FUNCTION_BLOCK RunAoiInspectionV1 EXTENDS RunUnitSlave
VAR_INPUT
	ngBinReady : BOOL;
	ngCounter : POINTER TO UDINT;
END_VAR
VAR_OUTPUT
END_VAR
VAR
	//devices
	ngCylinder : POINTER TO RunCylinder; // normal close cylinder
	
	aoiOut1Done AT%I* : BOOL ; //done
	aoiOut2Grade AT%I* : BOOL ; //ok/ng
	
	aoiTrigger AT%Q* : BOOL;
	//internal
	
	commIdTrigger AT%Q* : DWORD;
	
	//
	serialNGCounter : INT;
END_VAR
VAR PERSISTENT
	serialNGGoal AT%M* : INT ;
END_VAR
VAR CONSTANT
	ERR_CONSECUTIVE_NG : DWORD := 8001;
END_VAR

SUPER^();

CASE outputState OF
	//--------------------------------
	//	Initialization TODO, (Light on?)
	//--------------------------------	
	eSpecialStates.INITIAL_BEGIN:	
		bSerialTransition := ngCylinder^.Execute(eCylinderCommands.COMMAND_A);
		IF bSerialTransition THEN
			serialNGCounter := 0;
			aoiTrigger := FALSE;
		END_IF
	eSpecialStates.INITIAL_STATE_1:
		bSerialTransition := NOT aoiOut1Done;
		IF bSerialTransition THEN
			NextState := eSpecialStates.INITIAL_END;
		END_IF
	//---------------------------------
	//	Working
	//---------------------------------
	eSpecialStates.SLAVE_ENTER_PROCEDURE:
		// report id to SCADA?		
		transitionByte.0 := ngCylinder^.Execute(eCylinderCommands.COMMAND_A); //alway extend
		transitionByte.1 := NOT aoiOut1Done; //check aoi-done off
		
		//20200305 , aoi result would retained last status??
		//transitionByte.2 := NOT aoiOut2Grade; //check aoi-result as NG (fuse)
		
		bSerialTransition:= (transitionByte = 16#3);
	16#201:
		IF SlotBase^.Valid THEN
			aoiTrigger := TRUE; //set aoi-trigger on
			bSerialTransition := TRUE;
		ELSE
			//no material , leave	
			NextState := 16#205;
		END_IF
	16#202:
		bSerialTransition := aoiOut1Done;
	16#203:
		bSerialTransition := NOT aoiOut1Done;
		IF bSerialTransition THEN 
			commIdTrigger := SlotBase^.Id; //trigger the data logger
		END_IF
	16#204:
		//wait aoi-done on
		IF  NOT aoiOut2Grade THEN
			//-------------
			//	NG
			//-------------
			SlotBase^.Valid := FALSE; //set as inexsited
			bSerialTransition:=	ngBinReady;
			
			IF bSerialTransition THEN
				serialNGCounter := serialNGCounter+1;
				IF  serialNGCounter >=  serialNGGoal THEN
					THIS^.AlarmCode := ERR_CONSECUTIVE_NG;
					serialNGCounter := 0; //reset
				END_IF
				
				IF ngCounter<>0 THEN
					ngCounter^ := ngCounter^ +1; //count-up
				END_IF			
			END_IF
						
		ELSIF  aoiOut2Grade THEN
			//--------------
			//	OK 
			//--------------
			bSerialTransition := ngCylinder^.Execute(eCylinderCommands.COMMAND_B); //open gate
			IF bSerialTransition THEN
				serialNGCounter := 0; //reset
			END_IF
		ELSIF bIsBypassed THEN
			bSerialTransition:=	TRUE;
		else
			//--------------------------
			// wait until aoi_done raise
			//--------------------------
		END_IF
	16#205:
		aoiTrigger := FALSE; //reset
		
		IF NOT SlotBase^.Valid AND previousNode <>0 AND_THEN previousNode^.isPurged THEN
			isPurged := true; // i am purged
		END_IF
		
		
		NextState := eSpecialStates.SLAVE_WORK_DONE;
END_CASE

METHOD FB_init : BOOL
VAR_INPUT
	bInitRetains : BOOL; // if TRUE, the retain variables are initialized (warm start / cold start)
	bInCopyCode : BOOL;  // if TRUE, the instance afterwards gets moved into the copy code (online change)
	
	argParent : POINTER TO RunUnitGeneric;
	argSlotBase : POINTER TO RunMaterial;
	argSlotLast : POINTER TO RunMaterial;
	
	argWorkingSignal : POINTER TO BOOL;
	
	argNgCylinder : POINTER TO RunCylinder;
	
END_VAR
//initialize 
Parent := argParent;
SlotBase := argSlotBase;
SlotLast := argSlotLast;
//
IF bInitRetains THEN
	NextState := eSpecialStates.INITIAL_BEGIN;
END_IF

workingSignal := argWorkingSignal; //link

ngCylinder := argNgCylinder;
END_METHOD

END_FUNCTION_BLOCK

(* stored: Version 1.1.0.1, ProductVersion 3.1.4024.0
   POU RunAoiInspectionV1: Id {7255faf6-adcd-46ad-a421-c808180e9942}, SpecialFunc None
   Method FB_init: Id {0f87af46-5d5f-4c6d-b262-bc2c8522819a} *)
